ABB RAPID module: Module1.mod

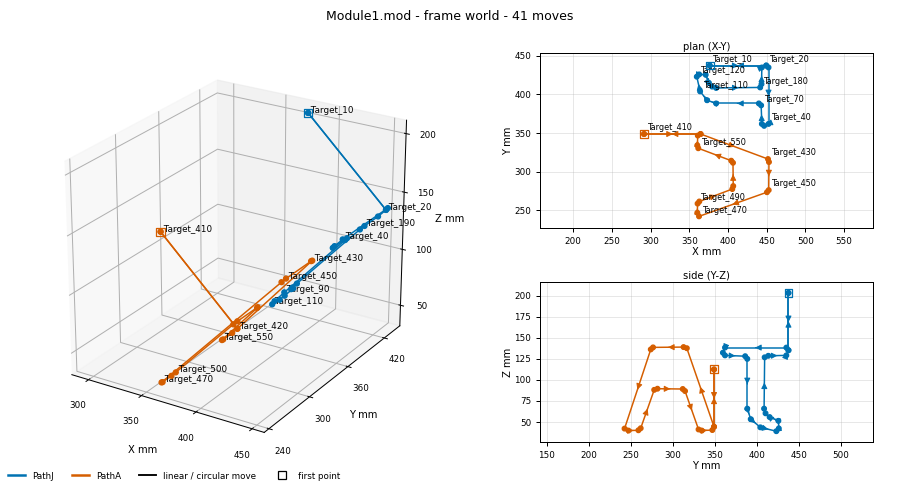
[picture p0: tool path of Module1.mod in frame world, 41 of 45 moves have a stored position in this frame; points joined in program order, loops and branches not executed]
MODULE Module1
        CONST robtarget Target_10:=[[47.084380669,72.82176413,-99.999847709],[0.707106718,0.000000835,-0.000000835,0.707106845],[0,0,0,0],[9E+09,9E+09,9E+09,9E+09,9E+09,9E+09]];
    CONST robtarget Target_20:=[[47.084380669,72.821528023,0.000152291],[0.707106718,0.000000835,-0.000000835,0.707106845],[0,0,0,0],[9E+09,9E+09,9E+09,9E+09,9E+09,9E+09]];
    CONST robtarget Target_30:=[[49.584380669,68.491401004,0.000142067],[0.707106718,0.000000835,-0.000000834,0.707106845],[0,0,0,0],[9E+09,9E+09,9E+09,9E+09,9E+09,9E+09]];
    CONST robtarget Target_40:=[[122.584380669,68.491401004,0.000142067],[0.707106718,0.000000834,-0.000000835,0.707106845],[0,0,0,0],[9E+09,9E+09,9E+09,9E+09,9E+09,9E+09]];
    CONST robtarget Target_50:=[[125.084380669,76.821528022,0.000161735],[0.707106718,0.000000835,-0.000000835,0.707106845],[0,0,0,0],[9E+09,9E+09,9E+09,9E+09,9E+09,9E+09]];
    CONST robtarget Target_60:=[[122.584380669,81.151655042,0.000171959],[0.707106718,0.000000835,-0.000000834,0.707106845],[0,0,0,0],[9E+09,9E+09,9E+09,9E+09,9E+09,9E+09]];
    CONST robtarget Target_70:=[[98.584380669,82.491401003,0.000175122],[0.707106718,0.000000835,-0.000000834,0.707106845],[0,0,0,0],[9E+09,9E+09,9E+09,9E+09,9E+09,9E+09]];
    CONST robtarget Target_80:=[[96.084380669,86.821528022,0.000185346],[0.707106718,0.000000835,-0.000000835,0.707106845],[0,0,0,0],[9E+09,9E+09,9E+09,9E+09,9E+09,9E+09]];
    CONST robtarget Target_90:=[[96.084380669,167.821528022,0.000376594],[0.707106718,0.000000835,-0.000000835,0.707106845],[0,0,0,0],[9E+09,9E+09,9E+09,9E+09,9E+09,9E+09]];
    CONST robtarget Target_100:=[[91.980477538,184.881916316,0.000416875],[0.707106718,0.000000834,-0.000000835,0.707106845],[0,0,0,0],[9E+09,9E+09,9E+09,9E+09,9E+09,9E+09]];
    CONST robtarget Target_110:=[[80.56669963,198.209502125,0.000448343],[0.707106718,0.000000835,-0.000000835,0.707106845],[0,0,0,0],[9E+09,9E+09,9E+09,9E+09,9E+09,9E+09]];
    CONST robtarget Target_120:=[[61.529602781,204.511779983,0.000463223],[0.707106718,0.000000834,-0.000000835,0.707106845],[0,0,0,0],[9E+09,9E+09,9E+09,9E+09,9E+09,9E+09]];
    CONST robtarget Target_130:=[[58.571449711,199.947696163,0.000452447],[0.707106718,0.000000835,-0.000000835,0.707106845],[0,0,0,0],[9E+09,9E+09,9E+09,9E+09,9E+09,9E+09]];
    CONST robtarget Target_140:=[[59.066921645,187.602126047,0.000423297],[0.707106718,0.000000835,-0.000000834,0.707106845],[0,0,0,0],[9E+09,9E+09,9E+09,9E+09,9E+09,9E+09]];
    CONST robtarget Target_150:=[[69.486591432,181.516871462,0.00040893],[0.707106718,0.000000835,-0.000000835,0.707106845],[0,0,0,0],[9E+09,9E+09,9E+09,9E+09,9E+09,9E+09]];
    CONST robtarget Target_160:=[[74.348947518,175.422403872,0.000394541],[0.707106718,0.000000835,-0.000000834,0.707106845],[0,0,0,0],[9E+09,9E+09,9E+09,9E+09,9E+09,9E+09]];
    CONST robtarget Target_170:=[[76.084380669,167.821528022,0.000376594],[0.707106718,0.000000835,-0.000000835,0.707106845],[0,0,0,0],[9E+09,9E+09,9E+09,9E+09,9E+09,9E+09]];
    CONST robtarget Target_180:=[[75.414507688,84.321528022,0.000179443],[0.707106718,0.000000834,-0.000000835,0.707106845],[0,0,0,0],[9E+09,9E+09,9E+09,9E+09,9E+09,9E+09]];
    CONST robtarget Target_190:=[[71.084380669,81.821528022,0.000173541],[0.707106718,0.000000835,-0.000000835,0.707106845],[0,0,0,0],[9E+09,9E+09,9E+09,9E+09,9E+09,9E+09]];
    CONST robtarget Target_200:=[[49.584380669,81.151655042,0.000171959],[0.707106718,0.000000834,-0.000000835,0.707106845],[0,0,0,0],[9E+09,9E+09,9E+09,9E+09,9E+09,9E+09]];
    CONST robtarget Target_210:=[[47.084380669,72.821528023,0.000152291],[0.707106718,0.000000835,-0.000000835,0.707106845],[0,0,0,0],[9E+09,9E+09,9E+09,9E+09,9E+09,9E+09]];
    CONST robtarget Target_220:=[[47.084380669,72.82176413,-99.999847709],[0.707106718,0.000000835,-0.000000835,0.707106845],[0,0,0,0],[9E+09,9E+09,9E+09,9E+09,9E+09,9E+09]];
    CONST robtarget Target_410:=[[135.654183782,197.290133375,-99.999553828],[0.707106718,0.000000835,-0.000000834,0.707106845],[0,-2,1,0],[9E+09,9E+09,9E+09,9E+09,9E+09,9E+09]];
    CONST robtarget Target_420:=[[135.654183782,197.289897267,0.000446171],[0.707106718,0.000000835,-0.000000834,0.707106845],[0,-2,1,0],[9E+09,9E+09,9E+09,9E+09,9E+09,9E+09]];
    CONST robtarget Target_430:=[[168.014089805,69.48895023,0.000144423],[0.707106718,0.000000835,-0.000000835,0.707106845],[0,-2,1,0],[9E+09,9E+09,9E+09,9E+09,9E+09,9E+09]];
    CONST robtarget Target_440:=[[171.881447769,67.658105066,0.0001401],[0.707106718,0.000000835,-0.000000835,0.707106845],[0,-2,1,0],[9E+09,9E+09,9E+09,9E+09,9E+09,9E+09]];
    CONST robtarget Target_450:=[[208.208010328,68.138936216,0.000141235],[0.707106718,0.000000834,-0.000000834,0.707106845],[0,-2,1,0],[9E+09,9E+09,9E+09,9E+09,9E+09,9E+09]];
    CONST robtarget Target_460:=[[210.920070135,71.448495589,0.00014905],[0.707106718,0.000000834,-0.000000835,0.707106845],[0,-2,1,0],[9E+09,9E+09,9E+09,9E+09,9E+09,9E+09]];
    CONST robtarget Target_470:=[[242.122624438,200.264159568,0.000453194],[0.707106718,0.000000834,-0.000000835,0.707106845],[0,-2,2,0],[9E+09,9E+09,9E+09,9E+09,9E+09,9E+09]];
    CONST robtarget Target_480:=[[237.444376859,203.499506745,0.000460832],[0.707106718,0.000000835,-0.000000835,0.707106845],[0,-2,2,0],[9E+09,9E+09,9E+09,9E+09,9E+09,9E+09]];
    CONST robtarget Target_490:=[[225.611094328,203.018675595,0.000459698],[0.707106718,0.000000834,-0.000000834,0.707106845],[0,-2,2,0],[9E+09,9E+09,9E+09,9E+09,9E+09,9E+09]];
    CONST robtarget Target_500:=[[222.899034521,199.709116223,0.000451884],[0.707106718,0.000000834,-0.000000835,0.707106845],[0,-2,2,0],[9E+09,9E+09,9E+09,9E+09,9E+09,9E+09]];
    CONST robtarget Target_510:=[[206.824866583,137.226696987,0.000304357],[0.707106718,0.000000835,-0.000000835,0.707106845],[0,-2,1,0],[9E+09,9E+09,9E+09,9E+09,9E+09,9E+09]];
    CONST robtarget Target_520:=[[202.95750862,135.395851823,0.000300034],[0.707106718,0.000000835,-0.000000835,0.707106845],[0,-2,1,0],[9E+09,9E+09,9E+09,9E+09,9E+09,9E+09]];
    CONST robtarget Target_530:=[[172.853111828,135.876682974,0.00030117],[0.707106718,0.000000834,-0.000000834,0.707106845],[0,-2,1,0],[9E+09,9E+09,9E+09,9E+09,9E+09,9E+09]];
    CONST robtarget Target_540:=[[170.141052021,139.186242346,0.000308984],[0.707106718,0.000000835,-0.000000834,0.707106845],[0,-2,1,0],[9E+09,9E+09,9E+09,9E+09,9E+09,9E+09]];
    CONST robtarget Target_550:=[[154.066884083,201.668661581,0.00045651],[0.707106718,0.000000835,-0.000000835,0.707106845],[0,-2,1,0],[9E+09,9E+09,9E+09,9E+09,9E+09,9E+09]];
    CONST robtarget Target_560:=[[150.19952612,203.499506745,0.000460832],[0.707106718,0.000000835,-0.000000835,0.707106845],[0,-2,1,0],[9E+09,9E+09,9E+09,9E+09,9E+09,9E+09]];
    CONST robtarget Target_570:=[[137.661656798,202.611882221,0.000458738],[0.707106718,0.000000835,-0.000000835,0.707106845],[0,-2,1,0],[9E+09,9E+09,9E+09,9E+09,9E+09,9E+09]];
    CONST robtarget Target_580:=[[135.654183782,197.289897267,0.000446171],[0.707106718,0.000000835,-0.000000834,0.707106845],[0,-2,1,0],[9E+09,9E+09,9E+09,9E+09,9E+09,9E+09]];
    CONST robtarget Target_590:=[[135.654183782,197.290133375,-99.999553828],[0.707106718,0.000000835,-0.000000834,0.707106845],[0,-2,1,0],[9E+09,9E+09,9E+09,9E+09,9E+09,9E+09]];
    CONST jointtarget Home:=[[0,0,0,0,0,0],[9E+09,9E+09,9E+09,9E+09,9E+09,9E+09]];
    CONST jointtarget JointTarget_2:=[[100,10,50,50,50,50],[9E+09,9E+09,9E+09,9E+09,9E+09,9E+09]];
    CONST jointtarget JointMID:=[[79.332642691,12.029773672,0,-35.09310633,46.732235952,0],[9E+09,9E+09,9E+09,9E+09,9E+09,9E+09]];
    CONST jointtarget TooLft:=[[82.050277404,0,0,-176.983209881,42.221418658,0],[9E+09,9E+09,9E+09,9E+09,9E+09,9E+09]];
    CONST jointtarget ToolRgt:=[[-90.591363032,0,-9.64451409,-176.983209881,42.221418658,0],[9E+09,9E+09,9E+09,9E+09,9E+09,9E+09]];
!***********************************************************
    !
    ! Module:  Module1
    !
    ! Description:
    !   <Insert description here>
    !
    ! Author: allan
    !
    ! Version: 1.0
    !
    !***********************************************************


    !***********************************************************
    !
    ! Procedure main
    !
    !   This is the entry point of your program
    !
    !***********************************************************
    PROC main()
        WaitDI DI_01,1;
        Homing;
        Set DO_01;
        WaitDI DI_02,1;
        Reset DO_01;
        Set DO_02;
        ToolLft;
        WaitDI DI_01,1;
        Reset DO_02;
        Set DO_01;
        Homing;
        WaitDI DI_03,1;
        Reset DO_01;
        Set DO_03;
        MidPoint;
        PathJ;
        PathA;
        MidPoint;
        WaitDI DI_01,1;
        Reset DO_03;
        Homing;
    ENDPROC
    PROC PathJ()
        MoveL Target_10,v150,fine,Dummy\WObj:=Tablero1;
        MoveL Target_20,v150,fine,Dummy\WObj:=Tablero1;
        MoveL Target_30,v150,fine,Dummy\WObj:=Tablero1;
        MoveL Target_40,v150,fine,Dummy\WObj:=Tablero1;
        MoveL Target_50,v150,fine,Dummy\WObj:=Tablero1;
        MoveL Target_60,v150,fine,Dummy\WObj:=Tablero1;
        MoveL Target_70,v150,fine,Dummy\WObj:=Tablero1;
        MoveL Target_80,v150,fine,Dummy\WObj:=Tablero1;
        MoveL Target_90,v150,fine,Dummy\WObj:=Tablero1;
        MoveL Target_100,v150,fine,Dummy\WObj:=Tablero1;
        MoveL Target_110,v150,fine,Dummy\WObj:=Tablero1;
        MoveL Target_120,v150,fine,Dummy\WObj:=Tablero1;
        MoveL Target_130,v150,fine,Dummy\WObj:=Tablero1;
        MoveL Target_140,v150,fine,Dummy\WObj:=Tablero1;
        MoveL Target_150,v150,fine,Dummy\WObj:=Tablero1;
        MoveL Target_160,v150,fine,Dummy\WObj:=Tablero1;
        MoveL Target_170,v150,fine,Dummy\WObj:=Tablero1;
        MoveL Target_180,v150,fine,Dummy\WObj:=Tablero1;
        MoveL Target_190,v150,fine,Dummy\WObj:=Tablero1;
        MoveL Target_200,v150,fine,Dummy\WObj:=Tablero1;
        MoveL Target_210,v150,fine,Dummy\WObj:=Tablero1;
        MoveL Target_220,v150,fine,Dummy\WObj:=Tablero1;
    ENDPROC
    PROC PathA()
        MoveL Target_410,v150,fine,Dummy\WObj:=Tablero1;
        MoveL Target_420,v150,fine,Dummy\WObj:=Tablero1;
        MoveL Target_430,v150,fine,Dummy\WObj:=Tablero1;
        MoveL Target_440,v150,fine,Dummy\WObj:=Tablero1;
        MoveL Target_450,v150,fine,Dummy\WObj:=Tablero1;
        MoveL Target_460,v150,fine,Dummy\WObj:=Tablero1;
        MoveL Target_470,v150,fine,Dummy\WObj:=Tablero1;
        MoveL Target_480,v150,fine,Dummy\WObj:=Tablero1;
        MoveL Target_490,v150,fine,Dummy\WObj:=Tablero1;
        MoveL Target_500,v150,fine,Dummy\WObj:=Tablero1;
        MoveL Target_510,v150,fine,Dummy\WObj:=Tablero1;
        MoveL Target_520,v150,fine,Dummy\WObj:=Tablero1;
        MoveL Target_530,v150,fine,Dummy\WObj:=Tablero1;
        MoveL Target_540,v150,fine,Dummy\WObj:=Tablero1;
        MoveL Target_550,v150,fine,Dummy\WObj:=Tablero1;
        MoveL Target_560,v150,fine,Dummy\WObj:=Tablero1;
        MoveL Target_570,v150,fine,Dummy\WObj:=Tablero1;
        MoveL Target_580,v150,fine,Dummy\WObj:=Tablero1;
        MoveL Target_590,v150,fine,Dummy\WObj:=Tablero1;
    ENDPROC
    PROC Homing()
        MoveAbsJ Home,v150,fine,Dummy\WObj:=Tablero1;
    ENDPROC
    PROC MidPoint()
        MoveAbsJ JointMID,v100,fine,MarcadorSR\WObj:=Tablero1;
    ENDPROC
    PROC ToolLft()
        MoveAbsJ TooLft,v150,fine,MarcadorSR\WObj:=Tablero1;
    ENDPROC
    PROC ToolRg()
        MoveAbsJ ToolRgt,v150,fine,MarcadorSR\WObj:=Tablero1;
    ENDPROC
ENDMODULE
